(*!
<summary>
Beckhoff EL1008_EX: Extended 8-channel digital input terminal with diagnostics.
</summary>
<description>
Extends EL1008 with EtherCAT Working Counter and slave state diagnostics. Note: Simple digital terminals do
not feature CoE mailbox, hence ADS address is not present.
When used for I/O, link located fields or their containing buffers to the matching selected PDOs.
The record is not a packed wire buffer; compiler padding is not part of the device specification.
Unlinked/default values do not prove valid I/O. The caller evaluates bus/channel validity before use.
Use one owner task per instance and externally synchronize other access; multi-field snapshots are not atomic.
Copies store data without creating hardware links. Keep borrowed field references valid while consumers are bound.
This passive record performs no validation, synchronization, configuration or protocol advancement.
WcState=TRUE means process-data exchange is invalid. State is acyclic EtherCAT/link information,
not proof of current measurement validity. Link diagnostics to the matching slave InfoData entries.
The selected PDO representation is documented by the base terminal model.
InputToggle signals an input update by changing state; TRUE alone does not mean fresh data.
</description>
*)
TYPE EL1008_EX EXTENDS EL1008 :
STRUCT
	WcState AT %I* : BOOL;
	InputToggle AT %I* : BOOL;
	State AT %I* : UINT;
END_STRUCT
END_TYPE

// ---- DigitalIO/Outputs/EL2809/EL2809.TcDUT
(*
SPDX-FileCopyrightText: © 2026 Oleksandr Tiutyk <trofimich@gmail.com>
SPDX-License-Identifier: MIT
License: https://opensource.org/license/mit
*)

(*!
<summary>
Beckhoff EL2809: 16-channel HD digital output terminal (24 V DC, 0.5 A).
</summary>
<description>
Process image mapping structure for the high-density EL2809 16-channel discrete 24 V DC 0.5 A output terminal.
When used for I/O, link located fields or their containing buffers to the matching selected PDOs.
The record is not a packed wire buffer; compiler padding is not part of the device specification.
Unlinked/default values do not prove valid I/O. The caller evaluates bus/channel validity before use.
Use one owner task per instance and externally synchronize other access; multi-field snapshots are not atomic.
Copies store data without creating hardware links. Keep borrowed field references valid while consumers are bound.
This passive record performs no validation, synchronization, configuration or protocol advancement.
</description>
*)
TYPE EL2809 :
STRUCT
	Ch01 AT %Q* : BOOL;
	Ch02 AT %Q* : BOOL;
	Ch03 AT %Q* : BOOL;
	Ch04 AT %Q* : BOOL;
	Ch05 AT %Q* : BOOL;
	Ch06 AT %Q* : BOOL;
	Ch07 AT %Q* : BOOL;
	Ch08 AT %Q* : BOOL;
	Ch09 AT %Q* : BOOL;
	Ch10 AT %Q* : BOOL;
	Ch11 AT %Q* : BOOL;
	Ch12 AT %Q* : BOOL;
	Ch13 AT %Q* : BOOL;
	Ch14 AT %Q* : BOOL;
	Ch15 AT %Q* : BOOL;
	Ch16 AT %Q* : BOOL;
END_STRUCT
END_TYPE

// ---- DigitalIO/Outputs/EL2809/EL2809_EX.TcDUT
(*
SPDX-FileCopyrightText: © 2026 Oleksandr Tiutyk <trofimich@gmail.com>
SPDX-License-Identifier: MIT
License: https://opensource.org/license/mit
*)

(*!
<summary>
Beckhoff EL2809_EX: Extended 16-channel HD digital output terminal with diagnostics.
</summary>
<description>
Extends EL2809 with EtherCAT Working Counter and slave state diagnostics.
When used for I/O, link located fields or their containing buffers to the matching selected PDOs.
The record is not a packed wire buffer; compiler padding is not part of the device specification.
Unlinked/default values do not prove valid I/O. The caller evaluates bus/channel validity before use.
Use one owner task per instance and externally synchronize other access; multi-field snapshots are not atomic.
Copies store data without creating hardware links. Keep borrowed field references valid while consumers are bound.
This passive record performs no validation, synchronization, configuration or protocol advancement.
WcState=TRUE means process-data exchange is invalid. State is acyclic EtherCAT/link information,
not proof of current measurement validity. Link diagnostics to the matching slave InfoData entries.
The selected PDO representation is documented by the base terminal model.
</description>
*)
TYPE EL2809_EX EXTENDS EL2809 :
STRUCT
	WcState AT %I* : BOOL;
	State AT %I* : UINT;
END_STRUCT
END_TYPE

// ---- DigitalIO/Outputs/EL2622/EL2622.TcDUT
(*
SPDX-FileCopyrightText: © 2026 Oleksandr Tiutyk <trofimich@gmail.com>
SPDX-License-Identifier: MIT
License: https://opensource.org/license/mit
*)

(*!
<summary>
Beckhoff EL2622: 2-channel relay output terminal (230 V AC / 30 V DC, normally open make contacts).
</summary>
<description>
Process image mapping structure for the EL2622 potential-free relay output terminal.
Each channel switches up to 5 A AC/DC for resistive loads or 2 A AC/DC for inductive loads.
The terminal has two make contacts, not changeover contacts, and does not pass through power contacts.
When used for I/O, link located fields or their containing buffers to the matching selected PDOs.
The record is not a packed wire buffer; compiler padding is not part of the device specification.
Unlinked/default values do not prove valid I/O. The caller evaluates bus/channel validity before use.
Use one owner task per instance and externally synchronize other access; multi-field snapshots are not atomic.
Copies store data without creating hardware links. Keep borrowed field references valid while consumers are bound.
This passive record performs no validation, synchronization, configuration or protocol advancement.
</description>
*)
TYPE EL2622 :
STRUCT
	Ch1 AT %Q* : BOOL;
	Ch2 AT %Q* : BOOL;
END_STRUCT
END_TYPE

// ---- DigitalIO/Outputs/EL2622/EL2622_EX.TcDUT
(*
SPDX-FileCopyrightText: © 2026 Oleksandr Tiutyk <trofimich@gmail.com>
SPDX-License-Identifier: MIT
License: https://opensource.org/license/mit
*)

(*!
<summary>
Beckhoff EL2622_EX: Extended 2-channel relay output terminal with diagnostics.
</summary>
<description>
Extends EL2622 with EtherCAT Working Counter and slave state diagnostics.
Two make contacts are rated 230 V AC / 30 V DC, with 5 A resistive or 2 A inductive current per channel.
When used for I/O, link located fields or their containing buffers to the matching selected PDOs.
The record is not a packed wire buffer; compiler padding is not part of the device specification.
Unlinked/default values do not prove valid I/O. The caller evaluates bus/channel validity before use.
Use one owner task per instance and externally synchronize other access; multi-field snapshots are not atomic.
Copies store data without creating hardware links. Keep borrowed field references valid while consumers are bound.
This passive record performs no validation, synchronization, configuration or protocol advancement.
WcState=TRUE means process-data exchange is invalid. State is acyclic EtherCAT/link information,
not proof of current measurement validity. Link diagnostics to the matching slave InfoData entries.
The selected PDO representation is documented by the base terminal model.
</description>
*)
TYPE EL2622_EX EXTENDS EL2622 :
STRUCT
	WcState AT %I* : BOOL;
	State AT %I* : UINT;
END_STRUCT
END_TYPE

// ---- DigitalIO/Outputs/EL2624/EL2624.TcDUT
(*
SPDX-FileCopyrightText: © 2026 Oleksandr Tiutyk <trofimich@gmail.com>
SPDX-License-Identifier: MIT
License: https://opensource.org/license/mit
*)

(*!
<summary>
Beckhoff EL2624: 4-channel relay output terminal (125 V AC / 30 V DC, normally open make contacts).
</summary>
<description>
Process image mapping structure for the EL2624 potential-free relay output terminal.
Resistive switching ratings are 0.5 A AC at 125 V AC and 2 A DC at 30 V DC per channel.
When used for I/O, link located fields or their containing buffers to the matching selected PDOs.
The record is not a packed wire buffer; compiler padding is not part of the device specification.
Unlinked/default values do not prove valid I/O. The caller evaluates bus/channel validity before use.
Use one owner task per instance and externally synchronize other access; multi-field snapshots are not atomic.
Copies store data without creating hardware links. Keep borrowed field references valid while consumers are bound.
This passive record performs no validation, synchronization, configuration or protocol advancement.
</description>
*)
TYPE EL2624 :
STRUCT
	Ch1 AT %Q* : BOOL;
	Ch2 AT %Q* : BOOL;
	Ch3 AT %Q* : BOOL;
	Ch4 AT %Q* : BOOL;
END_STRUCT
END_TYPE

// ---- DigitalIO/Outputs/EL2624/EL2624_EX.TcDUT
(*
SPDX-FileCopyrightText: © 2026 Oleksandr Tiutyk <trofimich@gmail.com>
SPDX-License-Identifier: MIT
License: https://opensource.org/license/mit
*)

(*!
<summary>
Beckhoff EL2624_EX: Extended 4-channel relay output terminal with diagnostics.
</summary>
<description>
Extends EL2624 with EtherCAT Working Counter and slave state diagnostics.
Four make contacts are rated 125 V AC / 30 V DC, with 0.5 A AC / 2 A DC resistive current per channel.
When used for I/O, link located fields or their containing buffers to the matching selected PDOs.
The record is not a packed wire buffer; compiler padding is not part of the device specification.
Unlinked/default values do not prove valid I/O. The caller evaluates bus/channel validity before use.
Use one owner task per instance and externally synchronize other access; multi-field snapshots are not atomic.
Copies store data without creating hardware links. Keep borrowed field references valid while consumers are bound.
This passive record performs no validation, synchronization, configuration or protocol advancement.
WcState=TRUE means process-data exchange is invalid. State is acyclic EtherCAT/link information,
not proof of current measurement validity. Link diagnostics to the matching slave InfoData entries.
The selected PDO representation is documented by the base terminal model.
</description>
*)
TYPE EL2624_EX EXTENDS EL2624 :
STRUCT
	WcState AT %I* : BOOL;
	State AT %I* : UINT;
END_STRUCT
END_TYPE

// ---- Serial/EL6001/EL6001.TcDUT
(*
SPDX-FileCopyrightText: © 2026 Oleksandr Tiutyk <trofimich@gmail.com>
SPDX-License-Identifier: MIT
License: https://opensource.org/license/mit
*)

(*!
<summary>
Beckhoff EL6001: 1-channel serial interface terminal (RS232).
</summary>
<description>
Process image mapping structure for the EL6001 1-channel RS232 communication terminal.
When used for I/O, link located fields or their containing buffers to the matching selected PDOs.
The record is not a packed wire buffer; compiler padding is not part of the device specification.
Unlinked/default values do not prove valid I/O. The caller evaluates bus/channel validity before use.
Use one owner task per instance and externally synchronize other access; multi-field snapshots are not atomic.
Copies store data without creating hardware links. Keep borrowed field references valid while consumers are bound.
This passive record performs no validation, synchronization, configuration or protocol advancement.
Select the 22-byte serial payload with 16-bit status/control words; larger buffers and 9-bit modes
are outside this model. The owning service implements the transmit/receive toggle handshake.
</description>
*)
TYPE EL6001 :
STRUCT
	Ch1 : EL6001_CHANNEL;
END_STRUCT
END_TYPE

// ---- Serial/EL6001/EL6001_CHANNEL.TcDUT
(*
SPDX-FileCopyrightText: © 2026 Oleksandr Tiutyk <trofimich@gmail.com>
SPDX-License-Identifier: MIT
License: https://opensource.org/license/mit
*)

(*!
<summary>
Beckhoff EL6001: Serial RS232 communication channel process image.
</summary>
<description>
Encapsulates 22-byte input (InData) and output (OutData) process data for the EL6001 RS232 interface.
When used for I/O, link located fields or their containing buffers to the matching selected PDOs.
The record is not a packed wire buffer; compiler padding is not part of the device specification.
Unlinked/default values do not prove valid I/O. The caller evaluates bus/channel validity before use.
Use one owner task per instance and externally synchronize other access; multi-field snapshots are not atomic.
Copies store data without creating hardware links. Keep borrowed field references valid while consumers are bound.
This passive record performs no validation, synchronization, configuration or protocol advancement.
Select the 22-byte serial payload with 16-bit status/control words; larger buffers and 9-bit modes
are outside this model. The owning service implements the transmit/receive toggle handshake.
</description>
*)
TYPE EL6001_CHANNEL :
STRUCT
	InData AT %I* : EL6xxx22ByteInData;
	OutData AT %Q* : EL6xxx22ByteOutData;
END_STRUCT
END_TYPE

// ---- Serial/EL6001/EL6001_EX.TcDUT
(*
SPDX-FileCopyrightText: © 2026 Oleksandr Tiutyk <trofimich@gmail.com>
SPDX-License-Identifier: MIT
License: https://opensource.org/license/mit
*)

(*!
<summary>
Beckhoff EL6001_EX: Extended 1-channel serial interface terminal with diagnostics.
</summary>
<description>
Extends EL6001 with EtherCAT Working Counter, slave state, and CoE mailbox ADS address diagnostics.
When used for I/O, link located fields or their containing buffers to the matching selected PDOs.
The record is not a packed wire buffer; compiler padding is not part of the device specification.
Unlinked/default values do not prove valid I/O. The caller evaluates bus/channel validity before use.
Use one owner task per instance and externally synchronize other access; multi-field snapshots are not atomic.
Copies store data without creating hardware links. Keep borrowed field references valid while consumers are bound.
This passive record performs no validation, synchronization, configuration or protocol advancement.
WcState=TRUE means process-data exchange is invalid. State is acyclic EtherCAT/link information,
not proof of current measurement validity. Link diagnostics to the matching slave InfoData entries.
The selected PDO representation is documented by the base terminal model.
InputToggle signals an input update by changing state; TRUE alone does not mean fresh data.
AdsAddr is acyclic mailbox addressing information, not a measurement-validity indicator.
Select the 22-byte serial payload with 16-bit status/control words; larger buffers and 9-bit modes
are outside this model. The owning service implements the transmit/receive toggle handshake.
</description>
*)
TYPE EL6001_EX EXTENDS EL6001 :
STRUCT
	WcState AT %I* : BOOL;
	InputToggle AT %I* : BOOL;
	State AT %I* : UINT;
	AdsAddr AT %I* : Global.AMSADDR;
END_STRUCT
END_TYPE

// ---- Serial/EL6002/EL6002.TcDUT
(*
SPDX-FileCopyrightText: © 2026 Oleksandr Tiutyk <trofimich@gmail.com>
SPDX-License-Identifier: MIT
License: https://opensource.org/license/mit
*)

(*!
<summary>
Beckhoff EL6002: 2-channel serial interface terminal (RS232).
</summary>
<description>
Process image mapping structure for the EL6002 2-channel RS232 communication terminal.
When used for I/O, link located fields or their containing buffers to the matching selected PDOs.
The record is not a packed wire buffer; compiler padding is not part of the device specification.
Unlinked/default values do not prove valid I/O. The caller evaluates bus/channel validity before use.
Use one owner task per instance and externally synchronize other access; multi-field snapshots are not atomic.
Copies store data without creating hardware links. Keep borrowed field references valid while consumers are bound.
This passive record performs no validation, synchronization, configuration or protocol advancement.
Select the 22-byte serial payload with 16-bit status/control words; larger buffers and 9-bit modes
are outside this model. The owning service implements the transmit/receive toggle handshake.
</description>
*)
TYPE EL6002 :
STRUCT
	Ch1 : EL6002_CHANNEL;
	Ch2 : EL6002_CHANNEL;
END_STRUCT
END_TYPE

// ---- Serial/EL6002/EL6002_CHANNEL.TcDUT
(*
SPDX-FileCopyrightText: © 2026 Oleksandr Tiutyk <trofimich@gmail.com>
SPDX-License-Identifier: MIT
License: https://opensource.org/license/mit
*)

(*!
<summary>
Beckhoff EL6002: Serial RS232 communication channel process image.
</summary>
<description>
Encapsulates 22-byte input (InData) and output (OutData) process data for the EL6002 RS232 interface.
When used for I/O, link located fields or their containing buffers to the matching selected PDOs.
The record is not a packed wire buffer; compiler padding is not part of the device specification.
Unlinked/default values do not prove valid I/O. The caller evaluates bus/channel validity before use.
Use one owner task per instance and externally synchronize other access; multi-field snapshots are not atomic.
Copies store data without creating hardware links. Keep borrowed field references valid while consumers are bound.
This passive record performs no validation, synchronization, configuration or protocol advancement.
Select the 22-byte serial payload with 16-bit status/control words; larger buffers and 9-bit modes
are outside this model. The owning service implements the transmit/receive toggle handshake.
</description>
*)
TYPE EL6002_CHANNEL :
STRUCT
	InData AT %I* : EL6xxx22ByteInData;
	OutData AT %Q* : EL6xxx22ByteOutData;
END_STRUCT
END_TYPE

// ---- Serial/EL6002/EL6002_EX.TcDUT
(*
SPDX-FileCopyrightText: © 2026 Oleksandr Tiutyk <trofimich@gmail.com>
SPDX-License-Identifier: MIT
License: https://opensource.org/license/mit
*)

(*!
<summary>
Beckhoff EL6002_EX: Extended 2-channel serial interface terminal with diagnostics.
</summary>
<description>
Extends EL6002 with EtherCAT Working Counter, slave state, and CoE mailbox ADS address diagnostics.
When used for I/O, link located fields or their containing buffers to the matching selected PDOs.
The record is not a packed wire buffer; compiler padding is not part of the device specification.
Unlinked/default values do not prove valid I/O. The caller evaluates bus/channel validity before use.
Use one owner task per instance and externally synchronize other access; multi-field snapshots are not atomic.
Copies store data without creating hardware links. Keep borrowed field references valid while consumers are bound.
This passive record performs no validation, synchronization, configuration or protocol advancement.
WcState=TRUE means process-data exchange is invalid. State is acyclic EtherCAT/link information,
not proof of current measurement validity. Link diagnostics to the matching slave InfoData entries.
The selected PDO representation is documented by the base terminal model.
InputToggle signals an input update by changing state; TRUE alone does not mean fresh data.
AdsAddr is acyclic mailbox addressing information, not a measurement-validity indicator.
Select the 22-byte serial payload with 16-bit status/control words; larger buffers and 9-bit modes
are outside this model. The owning service implements the transmit/receive toggle handshake.
</description>
*)
TYPE EL6002_EX EXTENDS EL6002 :
STRUCT
	WcState AT %I* : BOOL;
	InputToggle AT %I* : BOOL;
	State AT %I* : UINT;
	AdsAddr AT %I* : Global.AMSADDR;
END_STRUCT
END_TYPE

// ---- Serial/EL6021/EL6021.TcDUT
(*
SPDX-FileCopyrightText: © 2026 Oleksandr Tiutyk <trofimich@gmail.com>
SPDX-License-Identifier: MIT
License: https://opensource.org/license/mit
*)

(*!
<summary>
Beckhoff EL6021: 1-channel serial interface terminal (RS422 / RS485).
</summary>
<description>
Process image mapping structure for the EL6021 1-channel RS422/RS485 communication terminal.
When used for I/O, link located fields or their containing buffers to the matching selected PDOs.
The record is not a packed wire buffer; compiler padding is not part of the device specification.
Unlinked/default values do not prove valid I/O. The caller evaluates bus/channel validity before use.
Use one owner task per instance and externally synchronize other access; multi-field snapshots are not atomic.
Copies store data without creating hardware links. Keep borrowed field references valid while consumers are bound.
This passive record performs no validation, synchronization, configuration or protocol advancement.
Select the 22-byte serial payload with 16-bit status/control words; larger buffers and 9-bit modes
are outside this model. The owning service implements the transmit/receive toggle handshake.
</description>
*)
TYPE EL6021 :
STRUCT
	Ch1 : EL6021_CHANNEL;
END_STRUCT
END_TYPE

// ---- Serial/EL6021/EL6021_CHANNEL.TcDUT
(*
SPDX-FileCopyrightText: © 2026 Oleksandr Tiutyk <trofimich@gmail.com>
SPDX-License-Identifier: MIT
License: https://opensource.org/license/mit
*)

(*!
<summary>
Beckhoff EL6021: Serial RS422/RS485 communication channel process image.
</summary>
<description>
Encapsulates 22-byte input (InData) and output (OutData) process data for the EL6021 RS422/RS485 interface.
When used for I/O, link located fields or their containing buffers to the matching selected PDOs.
The record is not a packed wire buffer; compiler padding is not part of the device specification.
Unlinked/default values do not prove valid I/O. The caller evaluates bus/channel validity before use.
Use one owner task per instance and externally synchronize other access; multi-field snapshots are not atomic.
Copies store data without creating hardware links. Keep borrowed field references valid while consumers are bound.
This passive record performs no validation, synchronization, configuration or protocol advancement.
Select the 22-byte serial payload with 16-bit status/control words; larger buffers and 9-bit modes
are outside this model. The owning service implements the transmit/receive toggle handshake.
</description>
*)
TYPE EL6021_CHANNEL :
STRUCT
	InData AT %I* : EL6xxx22ByteInData;
	OutData AT %Q* : EL6xxx22ByteOutData;
END_STRUCT
END_TYPE

// ---- Serial/EL6021/EL6021_EX.TcDUT
(*
SPDX-FileCopyrightText: © 2026 Oleksandr Tiutyk <trofimich@gmail.com>
SPDX-License-Identifier: MIT
License: https://opensource.org/license/mit
*)

(*!
<summary>
Beckhoff EL6021_EX: Extended 1-channel serial interface terminal with diagnostics.
</summary>
<description>
Extends EL6021 with EtherCAT Working Counter, slave state, and CoE mailbox ADS address diagnostics.
When used for I/O, link located fields or their containing buffers to the matching selected PDOs.
The record is not a packed wire buffer; compiler padding is not part of the device specification.
Unlinked/default values do not prove valid I/O. The caller evaluates bus/channel validity before use.
Use one owner task per instance and externally synchronize other access; multi-field snapshots are not atomic.
Copies store data without creating hardware links. Keep borrowed field references valid while consumers are bound.
This passive record performs no validation, synchronization, configuration or protocol advancement.
WcState=TRUE means process-data exchange is invalid. State is acyclic EtherCAT/link information,
not proof of current measurement validity. Link diagnostics to the matching slave InfoData entries.
The selected PDO representation is documented by the base terminal model.
InputToggle signals an input update by changing state; TRUE alone does not mean fresh data.
AdsAddr is acyclic mailbox addressing information, not a measurement-validity indicator.
Select the 22-byte serial payload with 16-bit status/control words; larger buffers and 9-bit modes
are outside this model. The owning service implements the transmit/receive toggle handshake.
</description>
*)
TYPE EL6021_EX EXTENDS EL6021 :
STRUCT
	WcState AT %I* : BOOL;
	InputToggle AT %I* : BOOL;
	State AT %I* : UINT;
	AdsAddr AT %I* : Global.AMSADDR;
END_STRUCT
END_TYPE

// ---- Counters/COUNTER_INPUT_CHANNEL.TcDUT
(*
SPDX-FileCopyrightText: © 2026 Oleksandr Tiutyk <trofimich@gmail.com>
SPDX-License-Identifier: MIT
License: https://opensource.org/license/mit
*)

(*!
<summary>
Beckhoff counter input channel process image.
</summary>
<description>
Encapsulates 16-bit status word and 32-bit unsigned counter value (CounterValue : UDINT) for fast counter
terminals.
When used for I/O, link located fields or their containing buffers to the matching selected PDOs.
The record is not a packed wire buffer; compiler padding is not part of the device specification.
Unlinked/default values do not prove valid I/O. The caller evaluates bus/channel validity before use.
Use one owner task per instance and externally synchronize other access; multi-field snapshots are not atomic.
Copies store data without creating hardware links. Keep borrowed field references valid while consumers are bound.
This passive record performs no validation, synchronization, configuration or protocol advancement.
</description>
*)
TYPE COUNTER_INPUT_CHANNEL :
STRUCT
	Status AT %I* : WORD;
	CounterValue AT %I* : UDINT;
END_STRUCT
END_TYPE

// ---- Counters/COUNTER_OUTPUT_CHANNEL.TcDUT
(*
SPDX-FileCopyrightText: © 2026 Oleksandr Tiutyk <trofimich@gmail.com>
SPDX-License-Identifier: MIT
License: https://opensource.org/license/mit
*)

(*!
<summary>
Beckhoff counter output control channel process image.
</summary>
<description>
Encapsulates 16-bit control word and 32-bit unsigned preset counter value (SetCounterValue : UDINT) for fast
counter terminals.
When used for I/O, link located fields or their containing buffers to the matching selected PDOs.
The record is not a packed wire buffer; compiler padding is not part of the device specification.
Unlinked/default values do not prove valid I/O. The caller evaluates bus/channel validity before use.
Use one owner task per instance and externally synchronize other access; multi-field snapshots are not atomic.
Copies store data without creating hardware links. Keep borrowed field references valid while consumers are bound.
This passive record performs no validation, synchronization, configuration or protocol advancement.
</description>
*)
TYPE COUNTER_OUTPUT_CHANNEL :
STRUCT
	Control AT %Q* : WORD;
	SetCounterValue AT %Q* : UDINT;
END_STRUCT
END_TYPE

// ---- Counters/COUNTER_CHANNEL.TcDUT
(*
SPDX-FileCopyrightText: © 2026 Oleksandr Tiutyk <trofimich@gmail.com>
SPDX-License-Identifier: MIT
License: https://opensource.org/license/mit
*)

(*!
<summary>
Beckhoff bidirectional counter channel process image.
</summary>
<description>
Aggregates input status/value (COUNTER_INPUT_CHANNEL) and output control/preset (COUNTER_OUTPUT_CHANNEL) for
one counter channel.
When used for I/O, link located fields or their containing buffers to the matching selected PDOs.
The record is not a packed wire buffer; compiler padding is not part of the device specification.
Unlinked/default values do not prove valid I/O. The caller evaluates bus/channel validity before use.
Use one owner task per instance and externally synchronize other access; multi-field snapshots are not atomic.
Copies store data without creating hardware links. Keep borrowed field references valid while consumers are bound.
This passive record performs no validation, synchronization, configuration or protocol advancement.
</description>
*)
TYPE COUNTER_CHANNEL :
STRUCT
	In : COUNTER_INPUT_CHANNEL;
	Out : COUNTER_OUTPUT_CHANNEL;
END_STRUCT
END_TYPE

// ---- Counters/EL1502/EL1502.TcDUT
(*
SPDX-FileCopyrightText: © 2026 Oleksandr Tiutyk <trofimich@gmail.com>
SPDX-License-Identifier: MIT
License: https://opensource.org/license/mit
*)

(*!
<summary>
Beckhoff EL1502: 2-channel up/down counter terminal (24 V DC, 100 kHz).
</summary>
<description>
Requires the 2Ch. Counter assignment: TxPDOs 0x1A00/0x1A01 and RxPDOs 0x1600/0x1601.
Each channel is a 32-bit counter with 16-bit status/control; direction is configured through CoE.
The factory 1Ch. +/- Counter assignment 0x1A02/0x1602 is not represented.
This model does not provide two independent hardware up/down input pairs.
When used for I/O, link located fields or their containing buffers to the matching selected PDOs.
The record is not a packed wire buffer; compiler padding is not part of the device specification.
Unlinked/default values do not prove valid I/O. The caller evaluates bus/channel validity before use.
Use one owner task per instance and externally synchronize other access; multi-field snapshots are not atomic.
Copies store data without creating hardware links. Keep borrowed field references valid while consumers are bound.
This passive record performs no validation, synchronization, configuration or protocol advancement.
</description>
*)
TYPE EL1502 :
STRUCT
	Ch1 : COUNTER_CHANNEL;
	Ch2 : COUNTER_CHANNEL;
END_STRUCT
END_TYPE

// ---- Counters/EL1502/EL1502_EX.TcDUT
(*
SPDX-FileCopyrightText: © 2026 Oleksandr Tiutyk <trofimich@gmail.com>
SPDX-License-Identifier: MIT
License: https://opensource.org/license/mit
*)

(*!
<summary>
Beckhoff EL1502_EX: Extended 2-channel counter terminal with diagnostics.
</summary>
<description>
Extends EL1502 with EtherCAT Working Counter, slave state, and CoE mailbox ADS address diagnostics.
When used for I/O, link located fields or their containing buffers to the matching selected PDOs.
The record is not a packed wire buffer; compiler padding is not part of the device specification.
Unlinked/default values do not prove valid I/O. The caller evaluates bus/channel validity before use.
Use one owner task per instance and externally synchronize other access; multi-field snapshots are not atomic.
Copies store data without creating hardware links. Keep borrowed field references valid while consumers are bound.
This passive record performs no validation, synchronization, configuration or protocol advancement.
WcState=TRUE means process-data exchange is invalid. State is acyclic EtherCAT/link information,
not proof of current measurement validity. Link diagnostics to the matching slave InfoData entries.
The selected PDO representation is documented by the base terminal model.
InputToggle signals an input update by changing state; TRUE alone does not mean fresh data.
AdsAddr is acyclic mailbox addressing information, not a measurement-validity indicator.
</description>
*)
TYPE EL1502_EX EXTENDS EL1502 :
STRUCT
	WcState AT %I* : BOOL;
	InputToggle AT %I* : BOOL;
	State AT %I* : UINT;
	AdsAddr AT %I* : Global.AMSADDR;
END_STRUCT
END_TYPE

// ---- Counters/EL1512/EL1512.TcDUT
(*
SPDX-FileCopyrightText: © 2026 Oleksandr Tiutyk <trofimich@gmail.com>
SPDX-License-Identifier: MIT
License: https://opensource.org/license/mit
*)

(*!
<summary>
Beckhoff EL1512: 2-channel up/down counter terminal (24 V DC).
</summary>
<description>
Represents the default 2Ch. Counter assignment: TxPDOs 0x1A00/0x1A01 and RxPDOs 0x1600/0x1601.
Each channel has 16-bit status/control and a 32-bit counter/preset. Direction is configured through CoE.
Single-channel up/down or gated-counter assignments are outside this model.
When used for I/O, link located fields or their containing buffers to the matching selected PDOs.
The record is not a packed wire buffer; compiler padding is not part of the device specification.
Unlinked/default values do not prove valid I/O. The caller evaluates bus/channel validity before use.
Use one owner task per instance and externally synchronize other access; multi-field snapshots are not atomic.
Copies store data without creating hardware links. Keep borrowed field references valid while consumers are bound.
This passive record performs no validation, synchronization, configuration or protocol advancement.
</description>
*)
TYPE EL1512 :
STRUCT
	Ch1 : COUNTER_CHANNEL;
	Ch2 : COUNTER_CHANNEL;
END_STRUCT
END_TYPE

// ---- Counters/EL1512/EL1512_EX.TcDUT
(*
SPDX-FileCopyrightText: © 2026 Oleksandr Tiutyk <trofimich@gmail.com>
SPDX-License-Identifier: MIT
License: https://opensource.org/license/mit
*)

(*!
<summary>
Beckhoff EL1512_EX: Extended 2-channel counter terminal with diagnostics.
</summary>
<description>
Extends EL1512 with EtherCAT Working Counter, slave state, and CoE mailbox ADS address diagnostics.
When used for I/O, link located fields or their containing buffers to the matching selected PDOs.
The record is not a packed wire buffer; compiler padding is not part of the device specification.
Unlinked/default values do not prove valid I/O. The caller evaluates bus/channel validity before use.
Use one owner task per instance and externally synchronize other access; multi-field snapshots are not atomic.
Copies store data without creating hardware links. Keep borrowed field references valid while consumers are bound.
This passive record performs no validation, synchronization, configuration or protocol advancement.
WcState=TRUE means process-data exchange is invalid. State is acyclic EtherCAT/link information,
not proof of current measurement validity. Link diagnostics to the matching slave InfoData entries.
The selected PDO representation is documented by the base terminal model.
InputToggle signals an input update by changing state; TRUE alone does not mean fresh data.
AdsAddr is acyclic mailbox addressing information, not a measurement-validity indicator.
</description>
*)
TYPE EL1512_EX EXTENDS EL1512 :
STRUCT
	WcState AT %I* : BOOL;
	InputToggle AT %I* : BOOL;
	State AT %I* : UINT;
	AdsAddr AT %I* : Global.AMSADDR;
END_STRUCT
END_TYPE

// ---- Encoders/INCREMENTAL_ENCODER_INPUT_CHANNEL.TcDUT
(*
SPDX-FileCopyrightText: © 2026 Oleksandr Tiutyk <trofimich@gmail.com>
SPDX-License-Identifier: MIT
License: https://opensource.org/license/mit
*)

(*!
<summary>
Beckhoff incremental encoder input channel process image.
</summary>
<description>
Encapsulates 16-bit status word, 32-bit position value, and 32-bit captured latch value.
Use the matching 32-bit main PDO of EL5101 enhanced mode or EL5151. EL5152 has no latch and uses
INCREMENTAL_ENCODER_COUNTER_INPUT_CHANNEL instead; 16-bit process images are unsupported.
When used for I/O, link located fields or their containing buffers to the matching selected PDOs.
The record is not a packed wire buffer; compiler padding is not part of the device specification.
Unlinked/default values do not prove valid I/O. The caller evaluates bus/channel validity before use.
Use one owner task per instance and externally synchronize other access; multi-field snapshots are not atomic.
Copies store data without creating hardware links. Keep borrowed field references valid while consumers are bound.
This passive record performs no validation, synchronization, configuration or protocol advancement.
</description>
*)
TYPE INCREMENTAL_ENCODER_INPUT_CHANNEL :
STRUCT
	Status AT %I* : WORD;
	Value AT %I* : UDINT;
	Latch AT %I* : UDINT;
END_STRUCT
END_TYPE

// ---- Encoders/INCREMENTAL_ENCODER_OUTPUT_CHANNEL.TcDUT
(*
SPDX-FileCopyrightText: © 2026 Oleksandr Tiutyk <trofimich@gmail.com>
SPDX-License-Identifier: MIT
License: https://opensource.org/license/mit
*)

(*!
<summary>
Beckhoff incremental encoder output channel process image.
</summary>
<description>
Encapsulates 16-bit control word and 32-bit preset position value.
When used for I/O, link located fields or their containing buffers to the matching selected PDOs.
The record is not a packed wire buffer; compiler padding is not part of the device specification.
Unlinked/default values do not prove valid I/O. The caller evaluates bus/channel validity before use.
Use one owner task per instance and externally synchronize other access; multi-field snapshots are not atomic.
Copies store data without creating hardware links. Keep borrowed field references valid while consumers are bound.
This passive record performs no validation, synchronization, configuration or protocol advancement.
</description>
*)
TYPE INCREMENTAL_ENCODER_OUTPUT_CHANNEL :
STRUCT
	Control AT %Q* : WORD;
	SetValue AT %Q* : UDINT;
END_STRUCT
END_TYPE

// ---- Encoders/INCREMENTAL_ENCODER_CHANNEL.TcDUT
(*
SPDX-FileCopyrightText: © 2026 Oleksandr Tiutyk <trofimich@gmail.com>
SPDX-License-Identifier: MIT
License: https://opensource.org/license/mit
*)

(*!
<summary>
Beckhoff bidirectional incremental encoder channel process image.
</summary>
<description>
Aggregates input position/status/latch and output control/preset for an incremental encoder interface.
Requires the matching 32-bit EL5101 enhanced or EL5151 main PDOs. EL5152 uses the latch-free
INCREMENTAL_ENCODER_COUNTER_CHANNEL; do not substitute these channel types for each other.
When used for I/O, link located fields or their containing buffers to the matching selected PDOs.
The record is not a packed wire buffer; compiler padding is not part of the device specification.
Unlinked/default values do not prove valid I/O. The caller evaluates bus/channel validity before use.
Use one owner task per instance and externally synchronize other access; multi-field snapshots are not atomic.
Copies store data without creating hardware links. Keep borrowed field references valid while consumers are bound.
This passive record performs no validation, synchronization, configuration or protocol advancement.
</description>
*)
TYPE INCREMENTAL_ENCODER_CHANNEL :
STRUCT
	In : INCREMENTAL_ENCODER_INPUT_CHANNEL;
	Out : INCREMENTAL_ENCODER_OUTPUT_CHANNEL;
END_STRUCT
END_TYPE

// ---- Encoders/INCREMENTAL_ENCODER_COUNTER_INPUT_CHANNEL.TcDUT
(*
SPDX-FileCopyrightText: © 2026 Oleksandr Tiutyk <trofimich@gmail.com>
SPDX-License-Identifier: MIT
License: https://opensource.org/license/mit
*)

(*!
<summary>Beckhoff EL5152 32-bit incremental encoder feedback without a latch.</summary>
<description>
Represents the 32-bit main input PDO for one EL5152 channel (0x1A00 or 0x1A04).
Status is 16-bit; Value is the 32-bit counter. This terminal has no latch value.
Optional period/frequency PDOs are outside this channel; disable them or link them separately.
Link fields individually and evaluate bus/channel validity before use; unlinked zeros are not valid data.
Use one owner task and externally synchronize other access. Copies are not atomic multi-field snapshots.
When used for I/O, link located fields or their containing buffers to the matching selected PDOs.
The record is not a packed wire buffer; compiler padding is not part of the device specification.
Unlinked/default values do not prove valid I/O. The caller evaluates bus/channel validity before use.
Use one owner task per instance and externally synchronize other access; multi-field snapshots are not atomic.
Copies store data without creating hardware links. Keep borrowed field references valid while consumers are bound.
This passive record performs no validation, synchronization, configuration or protocol advancement.
</description>
*)
TYPE INCREMENTAL_ENCODER_COUNTER_INPUT_CHANNEL :
STRUCT
	Status AT %I* : WORD;
	Value AT %I* : UDINT;
END_STRUCT
END_TYPE

// ---- Encoders/INCREMENTAL_ENCODER_COUNTER_CHANNEL.TcDUT
(*
SPDX-FileCopyrightText: © 2026 Oleksandr Tiutyk <trofimich@gmail.com>
SPDX-License-Identifier: MIT
License: https://opensource.org/license/mit
*)

(*!
<summary>Beckhoff EL5152 32-bit incremental encoder channel without a latch.</summary>
<description>
Combines a latch-free 32-bit counter input with the 16-bit control word and 32-bit counter preset.
Select the 32-bit main PDOs for the corresponding EL5152 channel; optional period/frequency PDOs are separate.
Link input and output fields individually; the aggregate is not a packed EtherCAT packet.
Use one owner task; externally synchronize other access. Copies store data without creating hardware links.
When used for I/O, link located fields or their containing buffers to the matching selected PDOs.
The record is not a packed wire buffer; compiler padding is not part of the device specification.
Unlinked/default values do not prove valid I/O. The caller evaluates bus/channel validity before use.
Use one owner task per instance and externally synchronize other access; multi-field snapshots are not atomic.
Copies store data without creating hardware links. Keep borrowed field references valid while consumers are bound.
This passive record performs no validation, synchronization, configuration or protocol advancement.
</description>
*)
TYPE INCREMENTAL_ENCODER_COUNTER_CHANNEL :
STRUCT
	In : INCREMENTAL_ENCODER_COUNTER_INPUT_CHANNEL;
	Out : INCREMENTAL_ENCODER_OUTPUT_CHANNEL;
END_STRUCT
END_TYPE

// ---- Encoders/SSI_ENCODER_CHANNEL.TcDUT
(*
SPDX-FileCopyrightText: © 2026 Oleksandr Tiutyk <trofimich@gmail.com>
SPDX-License-Identifier: MIT
License: https://opensource.org/license/mit
*)

(*!
<summary>
Beckhoff SSI absolute encoder channel process image.
</summary>
<description>
Represents the SSI 32-bit position and two-byte status variant.
EL5001 requires firmware 11 or later and selection of the two-byte status PDO (0x1A01).
Earlier EL5001 firmware supports only one status byte and is incompatible with this channel.
For EL5002 select the corresponding two-byte status PDO for each channel. No byte-status conversion occurs.
When used for I/O, link located fields or their containing buffers to the matching selected PDOs.
The record is not a packed wire buffer; compiler padding is not part of the device specification.
Unlinked/default values do not prove valid I/O. The caller evaluates bus/channel validity before use.
Use one owner task per instance and externally synchronize other access; multi-field snapshots are not atomic.
Copies store data without creating hardware links. Keep borrowed field references valid while consumers are bound.
This passive record performs no validation, synchronization, configuration or protocol advancement.
</description>
*)
TYPE SSI_ENCODER_CHANNEL :
STRUCT
	Status AT %I* : WORD;
	Value AT %I* : UDINT;
END_STRUCT
END_TYPE

// ---- Encoders/EL5101/EL5101.TcDUT
(*
SPDX-FileCopyrightText: © 2026 Oleksandr Tiutyk <trofimich@gmail.com>
SPDX-License-Identifier: MIT
License: https://opensource.org/license/mit
*)

(*!
<summary>
Beckhoff EL5101: 1-channel incremental encoder interface terminal (RS422 / TTL, 5 V / 24 V).
</summary>
<description>
Requires enhanced operating mode, available on EL5101 from firmware 14 / hardware 09,
and Standard 32-bit (MDP 511): TxPDO 0x1A04 and RxPDO 0x1603.
Ch1 contains 16-bit status/control and 32-bit counter, latch and preset values.
The normal 16-bit mode and optional frequency/period/timestamp PDOs are outside this model.
When used for I/O, link located fields or their containing buffers to the matching selected PDOs.
The record is not a packed wire buffer; compiler padding is not part of the device specification.
Unlinked/default values do not prove valid I/O. The caller evaluates bus/channel validity before use.
Use one owner task per instance and externally synchronize other access; multi-field snapshots are not atomic.
Copies store data without creating hardware links. Keep borrowed field references valid while consumers are bound.
This passive record performs no validation, synchronization, configuration or protocol advancement.
</description>
*)
TYPE EL5101 :
STRUCT
	Ch1 : INCREMENTAL_ENCODER_CHANNEL;
END_STRUCT
END_TYPE

// ---- Encoders/EL5101/EL5101_EX.TcDUT
(*
SPDX-FileCopyrightText: © 2026 Oleksandr Tiutyk <trofimich@gmail.com>
SPDX-License-Identifier: MIT
License: https://opensource.org/license/mit
*)

(*!
<summary>
Beckhoff EL5101_EX: Extended 1-channel incremental encoder terminal with diagnostics.
</summary>
<description>
Extends EL5101 with EtherCAT Working Counter, slave state, and CoE mailbox ADS address diagnostics.
When used for I/O, link located fields or their containing buffers to the matching selected PDOs.
The record is not a packed wire buffer; compiler padding is not part of the device specification.
Unlinked/default values do not prove valid I/O. The caller evaluates bus/channel validity before use.
Use one owner task per instance and externally synchronize other access; multi-field snapshots are not atomic.
Copies store data without creating hardware links. Keep borrowed field references valid while consumers are bound.
This passive record performs no validation, synchronization, configuration or protocol advancement.
WcState=TRUE means process-data exchange is invalid. State is acyclic EtherCAT/link information,
not proof of current measurement validity. Link diagnostics to the matching slave InfoData entries.
The selected PDO representation is documented by the base terminal model.
InputToggle signals an input update by changing state; TRUE alone does not mean fresh data.
AdsAddr is acyclic mailbox addressing information, not a measurement-validity indicator.
</description>
*)
TYPE EL5101_EX EXTENDS EL5101 :
STRUCT
	WcState AT %I* : BOOL;
	InputToggle AT %I* : BOOL;
	State AT %I* : UINT;
	AdsAddr AT %I* : Global.AMSADDR;
END_STRUCT
END_TYPE

// ---- Encoders/EL5151/EL5151.TcDUT
(*
SPDX-FileCopyrightText: © 2026 Oleksandr Tiutyk <trofimich@gmail.com>
SPDX-License-Identifier: MIT
License: https://opensource.org/license/mit
*)

(*!
<summary>
Beckhoff EL5151: 1-channel incremental encoder interface terminal (24 V HTL, single-ended).
</summary>
<description>
Represents Standard 32-bit (MDP 511) main PDOs: TxPDO 0x1A00 and RxPDO 0x1600.
Ch1 contains 16-bit status/control and 32-bit counter, latch and preset values.
Optional period/frequency/timestamp PDOs are outside this model; disable or link them separately.
The Standard 16-bit process image is unsupported.
When used for I/O, link located fields or their containing buffers to the matching selected PDOs.
The record is not a packed wire buffer; compiler padding is not part of the device specification.
Unlinked/default values do not prove valid I/O. The caller evaluates bus/channel validity before use.
Use one owner task per instance and externally synchronize other access; multi-field snapshots are not atomic.
Copies store data without creating hardware links. Keep borrowed field references valid while consumers are bound.
This passive record performs no validation, synchronization, configuration or protocol advancement.
</description>
*)
TYPE EL5151 :
STRUCT
	Ch1 : INCREMENTAL_ENCODER_CHANNEL;
END_STRUCT
END_TYPE

// ---- Encoders/EL5151/EL5151_EX.TcDUT
(*
SPDX-FileCopyrightText: © 2026 Oleksandr Tiutyk <trofimich@gmail.com>
SPDX-License-Identifier: MIT
License: https://opensource.org/license/mit
*)

(*!
<summary>
Beckhoff EL5151_EX: Extended 1-channel 24 V incremental encoder terminal with diagnostics.
</summary>
<description>
Extends EL5151 with EtherCAT Working Counter, slave state, and CoE mailbox ADS address diagnostics.
When used for I/O, link located fields or their containing buffers to the matching selected PDOs.
The record is not a packed wire buffer; compiler padding is not part of the device specification.
Unlinked/default values do not prove valid I/O. The caller evaluates bus/channel validity before use.
Use one owner task per instance and externally synchronize other access; multi-field snapshots are not atomic.
Copies store data without creating hardware links. Keep borrowed field references valid while consumers are bound.
This passive record performs no validation, synchronization, configuration or protocol advancement.
WcState=TRUE means process-data exchange is invalid. State is acyclic EtherCAT/link information,
not proof of current measurement validity. Link diagnostics to the matching slave InfoData entries.
The selected PDO representation is documented by the base terminal model.
InputToggle signals an input update by changing state; TRUE alone does not mean fresh data.
AdsAddr is acyclic mailbox addressing information, not a measurement-validity indicator.
</description>
*)
TYPE EL5151_EX EXTENDS EL5151 :
STRUCT
	WcState AT %I* : BOOL;
	InputToggle AT %I* : BOOL;
	State AT %I* : UINT;
	AdsAddr AT %I* : Global.AMSADDR;
END_STRUCT
END_TYPE

// ---- Encoders/EL5152/EL5152.TcDUT
(*
SPDX-FileCopyrightText: © 2026 Oleksandr Tiutyk <trofimich@gmail.com>
SPDX-License-Identifier: MIT
License: https://opensource.org/license/mit
*)

(*!
<summary>
Beckhoff EL5152: 2-channel incremental encoder interface terminal (24 V HTL, single-ended).
</summary>
<description>
Represents the 32-bit main PDOs: channel 1 uses 0x1A00/0x1600; channel 2 uses 0x1A04/0x1602.
Both channels expose counter feedback and preset without a latch. Select Standard 32-bit (MDP 511);
optional period/frequency PDOs included by the ESI preset are outside this model and must be linked
separately if retained. The Standard 16-bit image is unsupported. Link each field individually.
Evaluate bus/channel validity before use. Use one owner task and synchronize other access.
When used for I/O, link located fields or their containing buffers to the matching selected PDOs.
The record is not a packed wire buffer; compiler padding is not part of the device specification.
Unlinked/default values do not prove valid I/O. The caller evaluates bus/channel validity before use.
Use one owner task per instance and externally synchronize other access; multi-field snapshots are not atomic.
Copies store data without creating hardware links. Keep borrowed field references valid while consumers are bound.
This passive record performs no validation, synchronization, configuration or protocol advancement.
</description>
*)
TYPE EL5152 :
STRUCT
	Ch1 : INCREMENTAL_ENCODER_COUNTER_CHANNEL;
	Ch2 : INCREMENTAL_ENCODER_COUNTER_CHANNEL;
END_STRUCT
END_TYPE

// ---- Encoders/EL5152/EL5152_EX.TcDUT
(*
SPDX-FileCopyrightText: © 2026 Oleksandr Tiutyk <trofimich@gmail.com>
SPDX-License-Identifier: MIT
License: https://opensource.org/license/mit
*)

(*!
<summary>
Beckhoff EL5152_EX: Extended 2-channel 24 V incremental encoder terminal with diagnostics.
</summary>
<description>
Extends EL5152 with EtherCAT Working Counter, slave state, and CoE mailbox ADS address diagnostics.
When used for I/O, link located fields or their containing buffers to the matching selected PDOs.
The record is not a packed wire buffer; compiler padding is not part of the device specification.
Unlinked/default values do not prove valid I/O. The caller evaluates bus/channel validity before use.
Use one owner task per instance and externally synchronize other access; multi-field snapshots are not atomic.
Copies store data without creating hardware links. Keep borrowed field references valid while consumers are bound.
This passive record performs no validation, synchronization, configuration or protocol advancement.
WcState=TRUE means process-data exchange is invalid. State is acyclic EtherCAT/link information,
not proof of current measurement validity. Link diagnostics to the matching slave InfoData entries.
The selected PDO representation is documented by the base terminal model.
InputToggle signals an input update by changing state; TRUE alone does not mean fresh data.
AdsAddr is acyclic mailbox addressing information, not a measurement-validity indicator.
</description>
*)
TYPE EL5152_EX EXTENDS EL5152 :
STRUCT
	WcState AT %I* : BOOL;
	InputToggle AT %I* : BOOL;
	State AT %I* : UINT;
	AdsAddr AT %I* : Global.AMSADDR;
END_STRUCT
END_TYPE

// ---- Encoders/EL5001/EL5001.TcDUT
(*
SPDX-FileCopyrightText: © 2026 Oleksandr Tiutyk <trofimich@gmail.com>
SPDX-License-Identifier: MIT
License: https://opensource.org/license/mit
*)

(*!
<summary>
Beckhoff EL5001: 1-channel SSI absolute encoder interface terminal.
</summary>
<description>
Process image mapping structure for the EL5001 synchronous serial interface (SSI) absolute encoder terminal.
Requires firmware 11 or later and the two-byte status PDO 0x1A01. The one-byte variant is unsupported.
When used for I/O, link located fields or their containing buffers to the matching selected PDOs.
The record is not a packed wire buffer; compiler padding is not part of the device specification.
Unlinked/default values do not prove valid I/O. The caller evaluates bus/channel validity before use.
Use one owner task per instance and externally synchronize other access; multi-field snapshots are not atomic.
Copies store data without creating hardware links. Keep borrowed field references valid while consumers are bound.
This passive record performs no validation, synchronization, configuration or protocol advancement.
</description>
*)
TYPE EL5001 :
STRUCT
	Ch1 : SSI_ENCODER_CHANNEL;
END_STRUCT
END_TYPE

// ---- Encoders/EL5001/EL5001_EX.TcDUT
(*
SPDX-FileCopyrightText: © 2026 Oleksandr Tiutyk <trofimich@gmail.com>
SPDX-License-Identifier: MIT
License: https://opensource.org/license/mit
*)

(*!
<summary>
Beckhoff EL5001_EX: Extended 1-channel SSI encoder terminal with diagnostics.
</summary>
<description>
Extends EL5001 with EtherCAT Working Counter, slave state, and CoE mailbox ADS address diagnostics.
When used for I/O, link located fields or their containing buffers to the matching selected PDOs.
The record is not a packed wire buffer; compiler padding is not part of the device specification.
Unlinked/default values do not prove valid I/O. The caller evaluates bus/channel validity before use.
Use one owner task per instance and externally synchronize other access; multi-field snapshots are not atomic.
Copies store data without creating hardware links. Keep borrowed field references valid while consumers are bound.
This passive record performs no validation, synchronization, configuration or protocol advancement.
WcState=TRUE means process-data exchange is invalid. State is acyclic EtherCAT/link information,
not proof of current measurement validity. Link diagnostics to the matching slave InfoData entries.
The selected PDO representation is documented by the base terminal model.
InputToggle signals an input update by changing state; TRUE alone does not mean fresh data.
AdsAddr is acyclic mailbox addressing information, not a measurement-validity indicator.
</description>
*)
TYPE EL5001_EX EXTENDS EL5001 :
STRUCT
	WcState AT %I* : BOOL;
	InputToggle AT %I* : BOOL;
	State AT %I* : UINT;
	AdsAddr AT %I* : Global.AMSADDR;
END_STRUCT
END_TYPE

// ---- Encoders/EL5002/EL5002.TcDUT
(*
SPDX-FileCopyrightText: © 2026 Oleksandr Tiutyk <trofimich@gmail.com>
SPDX-License-Identifier: MIT
License: https://opensource.org/license/mit
*)

(*!
<summary>
Beckhoff EL5002: 2-channel SSI absolute encoder interface terminal.
</summary>
<description>
Process image mapping structure for the EL5002 2-channel synchronous serial interface (SSI) absolute encoder
terminal.
Select the two-byte status PDO for each channel. The one-byte status variant is unsupported.
When used for I/O, link located fields or their containing buffers to the matching selected PDOs.
The record is not a packed wire buffer; compiler padding is not part of the device specification.
Unlinked/default values do not prove valid I/O. The caller evaluates bus/channel validity before use.
Use one owner task per instance and externally synchronize other access; multi-field snapshots are not atomic.
Copies store data without creating hardware links. Keep borrowed field references valid while consumers are bound.
This passive record performs no validation, synchronization, configuration or protocol advancement.
</description>
*)
TYPE EL5002 :
STRUCT
	Ch1 : SSI_ENCODER_CHANNEL;
	Ch2 : SSI_ENCODER_CHANNEL;
END_STRUCT
END_TYPE

// ---- Encoders/EL5002/EL5002_EX.TcDUT
(*
SPDX-FileCopyrightText: © 2026 Oleksandr Tiutyk <trofimich@gmail.com>
SPDX-License-Identifier: MIT
License: https://opensource.org/license/mit
*)

(*!
<summary>
Beckhoff EL5002_EX: Extended 2-channel SSI encoder terminal with diagnostics.
</summary>
<description>
Extends EL5002 with EtherCAT Working Counter, slave state, and CoE mailbox ADS address diagnostics.
When used for I/O, link located fields or their containing buffers to the matching selected PDOs.
The record is not a packed wire buffer; compiler padding is not part of the device specification.
Unlinked/default values do not prove valid I/O. The caller evaluates bus/channel validity before use.
Use one owner task per instance and externally synchronize other access; multi-field snapshots are not atomic.
Copies store data without creating hardware links. Keep borrowed field references valid while consumers are bound.
This passive record performs no validation, synchronization, configuration or protocol advancement.
WcState=TRUE means process-data exchange is invalid. State is acyclic EtherCAT/link information,
not proof of current measurement validity. Link diagnostics to the matching slave InfoData entries.
The selected PDO representation is documented by the base terminal model.
InputToggle signals an input update by changing state; TRUE alone does not mean fresh data.
AdsAddr is acyclic mailbox addressing information, not a measurement-validity indicator.
</description>
*)
TYPE EL5002_EX EXTENDS EL5002 :
STRUCT
	WcState AT %I* : BOOL;
	InputToggle AT %I* : BOOL;
	State AT %I* : UINT;
	AdsAddr AT %I* : Global.AMSADDR;
END_STRUCT
END_TYPE

// ---- PWM/PWM_OUTPUT_CHANNEL.TcDUT
(*
SPDX-FileCopyrightText: © 2026 Oleksandr Tiutyk <trofimich@gmail.com>
SPDX-License-Identifier: MIT
License: https://opensource.org/license/mit
*)

(*!
<summary>
Beckhoff PWM output channel process image.
</summary>
<description>
Represents the duty-only EL2502 standard PWM PDO with signed presentation selected through CoE.
DutyCycle 0..32767 represents 0..100 percent before user scaling; frequency is configured acyclically.
Cyclic-period and unsigned-presentation variants are outside this channel. No clamping or CoE configuration occurs.
When used for I/O, link located fields or their containing buffers to the matching selected PDOs.
The record is not a packed wire buffer; compiler padding is not part of the device specification.
Unlinked/default values do not prove valid I/O. The caller evaluates bus/channel validity before use.
Use one owner task per instance and externally synchronize other access; multi-field snapshots are not atomic.
Copies store data without creating hardware links. Keep borrowed field references valid while consumers are bound.
This passive record performs no validation, synchronization, configuration or protocol advancement.
</description>
*)
TYPE PWM_OUTPUT_CHANNEL :
STRUCT
	DutyCycle AT %Q* : INT;
END_STRUCT
END_TYPE

// ---- PWM/PULSE_TRAIN_INPUT_CHANNEL.TcDUT
(*
SPDX-FileCopyrightText: © 2026 Oleksandr Tiutyk <trofimich@gmail.com>
SPDX-License-Identifier: MIT
License: https://opensource.org/license/mit
*)

(*!
<summary>
Beckhoff pulse train output feedback status process image.
</summary>
<description>
Requires EL2521 Standard 32-bit (MDP 253/511), TxPDOs 0x1A01 and 0x1A05.
Status and CounterStatus belong to separate PDOs; both carry sync error at bit 13 and toggle at bit 15.
Status bit 6 reports a PTO error. Evaluate bus validity and both status words before using CounterValue.
Link each input field individually; zero values do not prove valid links. Legacy and 16-bit layouts are unsupported.
Use one owner task and externally synchronize other access; copies are not atomic multi-field snapshots.
When used for I/O, link located fields or their containing buffers to the matching selected PDOs.
The record is not a packed wire buffer; compiler padding is not part of the device specification.
Unlinked/default values do not prove valid I/O. The caller evaluates bus/channel validity before use.
Use one owner task per instance and externally synchronize other access; multi-field snapshots are not atomic.
Copies store data without creating hardware links. Keep borrowed field references valid while consumers are bound.
This passive record performs no validation, synchronization, configuration or protocol advancement.
</description>
*)
TYPE PULSE_TRAIN_INPUT_CHANNEL :
STRUCT
	Status AT %I* : WORD;
	//! <summary>ENC status from 0x1A05: counter-set acknowledgement bit 2, underflow 3 and overflow 4.</summary>
	CounterStatus AT %I* : WORD;
	//! <summary>32-bit feedback at 0x6020:11 from ENC Status PDO 0x1A05.</summary>
	CounterValue AT %I* : UDINT;
END_STRUCT
END_TYPE

// ---- PWM/PULSE_TRAIN_OUTPUT_CHANNEL.TcDUT
(*
SPDX-FileCopyrightText: © 2026 Oleksandr Tiutyk <trofimich@gmail.com>
SPDX-License-Identifier: MIT
License: https://opensource.org/license/mit
*)

(*!
<summary>
Beckhoff pulse train output command process image.
</summary>
<description>
Requires EL2521 enhanced mode, Standard 32-bit (MDP 253/511): RxPDOs 0x1601, 0x1607 and 0x1605.
Control bits 0, 1 and 2 select the base frequency, disable the ramp and start target travel.
Frequency preserves the UINT16 PDO bit pattern, including direction encoding selected through CoE.
In relative mode the interpreted command scales the selected base frequency by 1/32767; in direct mode
CoE 0x8010:16 multiplies the interpreted command in 0.01 Hz units. Frequency is not a 32-bit Hz value.
TargetCounterValue is a separate 32-bit target; SetCounterValue presets encoder feedback.
Link fields individually; this aggregate is not a packed wire buffer. Configure CoE before enabling outputs.
Use one owner task; externally synchronize other access. Copies do not create links or an atomic snapshot.
When used for I/O, link located fields or their containing buffers to the matching selected PDOs.
The record is not a packed wire buffer; compiler padding is not part of the device specification.
Unlinked/default values do not prove valid I/O. The caller evaluates bus/channel validity before use.
Use one owner task per instance and externally synchronize other access; multi-field snapshots are not atomic.
Copies store data without creating hardware links. Keep borrowed field references valid while consumers are bound.
This passive record performs no validation, synchronization, configuration or protocol advancement.
</description>
*)
TYPE PULSE_TRAIN_OUTPUT_CHANNEL :
STRUCT
	Control AT %Q* : WORD;
	//! <summary>Raw frequency command at 0x7010:11; interpretation follows CoE scaling and sign representation.</summary>
	Frequency AT %Q* : UINT;
	//! <summary>32-bit target at 0x7010:12, transmitted by PTO Target PDO 0x1607.</summary>
	TargetCounterValue AT %Q* : UDINT;
	//! <summary>ENC control from PDO 0x1605; bit 2 requests setting the feedback counter.</summary>
	CounterControl AT %Q* : WORD;
	//! <summary>Counter preset at 0x7020:11, accepted through CounterControl bit 2.</summary>
	SetCounterValue AT %Q* : UDINT;
END_STRUCT
END_TYPE

// ---- PWM/PULSE_TRAIN_CHANNEL.TcDUT
(*
SPDX-FileCopyrightText: © 2026 Oleksandr Tiutyk <trofimich@gmail.com>
SPDX-License-Identifier: MIT
License: https://opensource.org/license/mit
*)

(*!
<summary>
Beckhoff bidirectional pulse train channel process image.
</summary>
<description>
Combines EL2521 Standard 32-bit (MDP 253/511) input and output endpoints.
Select TxPDOs 0x1A01/0x1A05 and RxPDOs 0x1601/0x1607/0x1605 in enhanced operating mode.
Includes a 16-bit frequency command, 32-bit target, counter feedback and counter preset.
Link input and output fields individually; the aggregate is not one contiguous EtherCAT packet.
Use one owner task; synchronize external access. Copying stores data without creating new hardware links.
When used for I/O, link located fields or their containing buffers to the matching selected PDOs.
The record is not a packed wire buffer; compiler padding is not part of the device specification.
Unlinked/default values do not prove valid I/O. The caller evaluates bus/channel validity before use.
Use one owner task per instance and externally synchronize other access; multi-field snapshots are not atomic.
Copies store data without creating hardware links. Keep borrowed field references valid while consumers are bound.
This passive record performs no validation, synchronization, configuration or protocol advancement.
</description>
*)
TYPE PULSE_TRAIN_CHANNEL :
STRUCT
	In : PULSE_TRAIN_INPUT_CHANNEL;
	Out : PULSE_TRAIN_OUTPUT_CHANNEL;
END_STRUCT
END_TYPE

// ---- PWM/EL2502/EL2502.TcDUT
(*
SPDX-FileCopyrightText: © 2026 Oleksandr Tiutyk <trofimich@gmail.com>
SPDX-License-Identifier: MIT
License: https://opensource.org/license/mit
*)

(*!
<summary>
Beckhoff EL2502: 2-channel PWM output terminal (24 V DC, up to 20 kHz).
</summary>
<description>
Requires the duty-only Pulse width (standard) assignment, RxPDOs 0x1600 and 0x1601,
with signed presentation selected through CoE. Configure period/frequency before enabling outputs.
Cyclic-period and unsigned-presentation variants are outside this model.
When used for I/O, link located fields or their containing buffers to the matching selected PDOs.
The record is not a packed wire buffer; compiler padding is not part of the device specification.
Unlinked/default values do not prove valid I/O. The caller evaluates bus/channel validity before use.
Use one owner task per instance and externally synchronize other access; multi-field snapshots are not atomic.
Copies store data without creating hardware links. Keep borrowed field references valid while consumers are bound.
This passive record performs no validation, synchronization, configuration or protocol advancement.
</description>
*)
TYPE EL2502 :
STRUCT
	Ch1 : PWM_OUTPUT_CHANNEL;
	Ch2 : PWM_OUTPUT_CHANNEL;
END_STRUCT
END_TYPE

// ---- PWM/EL2502/EL2502_EX.TcDUT
(*
SPDX-FileCopyrightText: © 2026 Oleksandr Tiutyk <trofimich@gmail.com>
SPDX-License-Identifier: MIT
License: https://opensource.org/license/mit
*)

(*!
<summary>
Beckhoff EL2502_EX: Extended 2-channel PWM output terminal with diagnostics.
</summary>
<description>
Extends EL2502 with EtherCAT Working Counter, slave state, and CoE mailbox ADS address diagnostics. Note:
Output terminal does not feature InputToggle.
When used for I/O, link located fields or their containing buffers to the matching selected PDOs.
The record is not a packed wire buffer; compiler padding is not part of the device specification.
Unlinked/default values do not prove valid I/O. The caller evaluates bus/channel validity before use.
Use one owner task per instance and externally synchronize other access; multi-field snapshots are not atomic.
Copies store data without creating hardware links. Keep borrowed field references valid while consumers are bound.
This passive record performs no validation, synchronization, configuration or protocol advancement.
WcState=TRUE means process-data exchange is invalid. State is acyclic EtherCAT/link information,
not proof of current measurement validity. Link diagnostics to the matching slave InfoData entries.
The selected PDO representation is documented by the base terminal model.
AdsAddr is acyclic mailbox addressing information, not a measurement-validity indicator.
</description>
*)
TYPE EL2502_EX EXTENDS EL2502 :
STRUCT
	WcState AT %I* : BOOL;
	State AT %I* : UINT;
	AdsAddr AT %I* : Global.AMSADDR;
END_STRUCT
END_TYPE

// ---- PWM/EL2521/EL2521.TcDUT
(*
SPDX-FileCopyrightText: © 2026 Oleksandr Tiutyk <trofimich@gmail.com>
SPDX-License-Identifier: MIT
License: https://opensource.org/license/mit
*)

(*!
<summary>
Beckhoff EL2521: 1-channel pulse train output terminal (pulse/direction, up to 500 kHz).
</summary>
<description>
Requires enhanced operating mode (firmware 03 / hardware 02 or later supporting this preset)
and Predefined PDO Assignment Standard 32-bit (MDP 253/511).
Ch1 covers TxPDOs 0x1A01/0x1A05 and RxPDOs 0x1601/0x1607/0x1605.
Frequency remains a raw 16-bit command; target, counter feedback and counter preset are 32-bit.
Legacy and Standard 16-bit images are unsupported. Link each field separately and evaluate input validity.
Use one owner task; externally synchronize other access. Copies are data, not new links or atomic snapshots.
When used for I/O, link located fields or their containing buffers to the matching selected PDOs.
The record is not a packed wire buffer; compiler padding is not part of the device specification.
Unlinked/default values do not prove valid I/O. The caller evaluates bus/channel validity before use.
Use one owner task per instance and externally synchronize other access; multi-field snapshots are not atomic.
Copies store data without creating hardware links. Keep borrowed field references valid while consumers are bound.
This passive record performs no validation, synchronization, configuration or protocol advancement.
</description>
*)
TYPE EL2521 :
STRUCT
	Ch1 : PULSE_TRAIN_CHANNEL;
END_STRUCT
END_TYPE

// ---- PWM/EL2521/EL2521_EX.TcDUT
(*
SPDX-FileCopyrightText: © 2026 Oleksandr Tiutyk <trofimich@gmail.com>
SPDX-License-Identifier: MIT
License: https://opensource.org/license/mit
*)

(*!
<summary>
Beckhoff EL2521_EX: Extended 1-channel pulse train terminal with diagnostics.
</summary>
<description>
Extends EL2521 with EtherCAT Working Counter, slave state, and CoE mailbox ADS address diagnostics.
When used for I/O, link located fields or their containing buffers to the matching selected PDOs.
The record is not a packed wire buffer; compiler padding is not part of the device specification.
Unlinked/default values do not prove valid I/O. The caller evaluates bus/channel validity before use.
Use one owner task per instance and externally synchronize other access; multi-field snapshots are not atomic.
Copies store data without creating hardware links. Keep borrowed field references valid while consumers are bound.
This passive record performs no validation, synchronization, configuration or protocol advancement.
WcState=TRUE means process-data exchange is invalid. State is acyclic EtherCAT/link information,
not proof of current measurement validity. Link diagnostics to the matching slave InfoData entries.
The selected PDO representation is documented by the base terminal model.
InputToggle signals an input update by changing state; TRUE alone does not mean fresh data.
AdsAddr is acyclic mailbox addressing information, not a measurement-validity indicator.
</description>
*)
TYPE EL2521_EX EXTENDS EL2521 :
STRUCT
	WcState AT %I* : BOOL;
	InputToggle AT %I* : BOOL;
	State AT %I* : UINT;
	AdsAddr AT %I* : Global.AMSADDR;
END_STRUCT
END_TYPE

// ---- AnalogIO/Inputs/EL3051/EL3051.TcDUT
(*
SPDX-FileCopyrightText: © 2026 Oleksandr Tiutyk <trofimich@gmail.com>
SPDX-License-Identifier: MIT
License: https://opensource.org/license/mit
*)

(*!
<summary>
Beckhoff EL3051: 1-channel analog input terminal (4 .. 20 mA, 12-bit single-ended).
</summary>
<description>
Process image mapping structure for the EL3051 EtherCAT terminal with 1 analog input channel(s).
When used for I/O, link located fields or their containing buffers to the matching selected PDOs.
The record is not a packed wire buffer; compiler padding is not part of the device specification.
Unlinked/default values do not prove valid I/O. The caller evaluates bus/channel validity before use.
Use one owner task per instance and externally synchronize other access; multi-field snapshots are not atomic.
Copies store data without creating hardware links. Keep borrowed field references valid while consumers are bound.
This passive record performs no validation, synchronization, configuration or protocol advancement.
Select standard status-plus-value PDOs matching the declared Value type; compact value-only PDOs
are outside this model. Configure electrical range and scaling separately on the device.
</description>
*)
TYPE EL3051 :
STRUCT
	Ch1 : ANALOG_INPUT_INT_CHANNEL;
END_STRUCT
END_TYPE

// ---- AnalogIO/Inputs/EL3051/EL3051_EX.TcDUT
(*
SPDX-FileCopyrightText: © 2026 Oleksandr Tiutyk <trofimich@gmail.com>
SPDX-License-Identifier: MIT
License: https://opensource.org/license/mit
*)

(*!
<summary>
Beckhoff EL3051_EX: Extended 1-channel analog input terminal (4 .. 20 mA, 12-bit single-ended) with
diagnostics.
</summary>
<description>
Extends EL3051 with EtherCAT Working Counter, slave state, and CoE mailbox ADS address diagnostics.
When used for I/O, link located fields or their containing buffers to the matching selected PDOs.
The record is not a packed wire buffer; compiler padding is not part of the device specification.
Unlinked/default values do not prove valid I/O. The caller evaluates bus/channel validity before use.
Use one owner task per instance and externally synchronize other access; multi-field snapshots are not atomic.
Copies store data without creating hardware links. Keep borrowed field references valid while consumers are bound.
This passive record performs no validation, synchronization, configuration or protocol advancement.
WcState=TRUE means process-data exchange is invalid. State is acyclic EtherCAT/link information,
not proof of current measurement validity. Link diagnostics to the matching slave InfoData entries.
The selected PDO representation is documented by the base terminal model.
InputToggle signals an input update by changing state; TRUE alone does not mean fresh data.
AdsAddr is acyclic mailbox addressing information, not a measurement-validity indicator.
Select standard status-plus-value PDOs matching the declared Value type; compact value-only PDOs
are outside this model. Configure electrical range and scaling separately on the device.
</description>
*)
TYPE EL3051_EX EXTENDS EL3051 :
STRUCT
	WcState AT %I* : BOOL;
	InputToggle AT %I* : BOOL;
	State AT %I* : UINT;
	AdsAddr AT %I* : Global.AMSADDR;
END_STRUCT
END_TYPE

// ---- AnalogIO/Inputs/EL3052/EL3052.TcDUT
(*
SPDX-FileCopyrightText: © 2026 Oleksandr Tiutyk <trofimich@gmail.com>
SPDX-License-Identifier: MIT
License: https://opensource.org/license/mit
*)

(*!
<summary>
Beckhoff EL3052: 2-channel analog input terminal (4 .. 20 mA, 12-bit single-ended).
</summary>
<description>
Process image mapping structure for the EL3052 EtherCAT terminal with 2 analog input channel(s).
When used for I/O, link located fields or their containing buffers to the matching selected PDOs.
The record is not a packed wire buffer; compiler padding is not part of the device specification.
Unlinked/default values do not prove valid I/O. The caller evaluates bus/channel validity before use.
Use one owner task per instance and externally synchronize other access; multi-field snapshots are not atomic.
Copies store data without creating hardware links. Keep borrowed field references valid while consumers are bound.
This passive record performs no validation, synchronization, configuration or protocol advancement.
Select standard status-plus-value PDOs matching the declared Value type; compact value-only PDOs
are outside this model. Configure electrical range and scaling separately on the device.
</description>
*)
TYPE EL3052 :
STRUCT
	Ch1 : ANALOG_INPUT_INT_CHANNEL;
	Ch2 : ANALOG_INPUT_INT_CHANNEL;
END_STRUCT
END_TYPE

// ---- AnalogIO/Inputs/EL3052/EL3052_EX.TcDUT
(*
SPDX-FileCopyrightText: © 2026 Oleksandr Tiutyk <trofimich@gmail.com>
SPDX-License-Identifier: MIT
License: https://opensource.org/license/mit
*)

(*!
<summary>
Beckhoff EL3052_EX: Extended 2-channel analog input terminal (4 .. 20 mA, 12-bit single-ended) with
diagnostics.
</summary>
<description>
Extends EL3052 with EtherCAT Working Counter, slave state, and CoE mailbox ADS address diagnostics.
When used for I/O, link located fields or their containing buffers to the matching selected PDOs.
The record is not a packed wire buffer; compiler padding is not part of the device specification.
Unlinked/default values do not prove valid I/O. The caller evaluates bus/channel validity before use.
Use one owner task per instance and externally synchronize other access; multi-field snapshots are not atomic.
Copies store data without creating hardware links. Keep borrowed field references valid while consumers are bound.
This passive record performs no validation, synchronization, configuration or protocol advancement.
WcState=TRUE means process-data exchange is invalid. State is acyclic EtherCAT/link information,
not proof of current measurement validity. Link diagnostics to the matching slave InfoData entries.
The selected PDO representation is documented by the base terminal model.
InputToggle signals an input update by changing state; TRUE alone does not mean fresh data.
AdsAddr is acyclic mailbox addressing information, not a measurement-validity indicator.
Select standard status-plus-value PDOs matching the declared Value type; compact value-only PDOs
are outside this model. Configure electrical range and scaling separately on the device.
</description>
*)
TYPE EL3052_EX EXTENDS EL3052 :
STRUCT
	WcState AT %I* : BOOL;
	InputToggle AT %I* : BOOL;
	State AT %I* : UINT;
	AdsAddr AT %I* : Global.AMSADDR;
END_STRUCT
END_TYPE

// ---- AnalogIO/Inputs/EL3054/EL3054.TcDUT
(*
SPDX-FileCopyrightText: © 2026 Oleksandr Tiutyk <trofimich@gmail.com>
SPDX-License-Identifier: MIT
License: https://opensource.org/license/mit
*)

(*!
<summary>
Beckhoff EL3054: 4-channel analog input terminal (4 .. 20 mA, 12-bit single-ended).
</summary>
<description>
Process image mapping structure for the EL3054 EtherCAT terminal with 4 analog input channel(s).
When used for I/O, link located fields or their containing buffers to the matching selected PDOs.
The record is not a packed wire buffer; compiler padding is not part of the device specification.
Unlinked/default values do not prove valid I/O. The caller evaluates bus/channel validity before use.
Use one owner task per instance and externally synchronize other access; multi-field snapshots are not atomic.
Copies store data without creating hardware links. Keep borrowed field references valid while consumers are bound.
This passive record performs no validation, synchronization, configuration or protocol advancement.
Select standard status-plus-value PDOs matching the declared Value type; compact value-only PDOs
are outside this model. Configure electrical range and scaling separately on the device.
</description>
*)
TYPE EL3054 :
STRUCT
	Ch1 : ANALOG_INPUT_INT_CHANNEL;
	Ch2 : ANALOG_INPUT_INT_CHANNEL;
	Ch3 : ANALOG_INPUT_INT_CHANNEL;
	Ch4 : ANALOG_INPUT_INT_CHANNEL;
END_STRUCT
END_TYPE

// ---- AnalogIO/Inputs/EL3054/EL3054_EX.TcDUT
(*
SPDX-FileCopyrightText: © 2026 Oleksandr Tiutyk <trofimich@gmail.com>
SPDX-License-Identifier: MIT
License: https://opensource.org/license/mit
*)

(*!
<summary>
Beckhoff EL3054_EX: Extended 4-channel analog input terminal (4 .. 20 mA, 12-bit single-ended) with
diagnostics.
</summary>
<description>
Extends EL3054 with EtherCAT Working Counter, slave state, and CoE mailbox ADS address diagnostics.
When used for I/O, link located fields or their containing buffers to the matching selected PDOs.
The record is not a packed wire buffer; compiler padding is not part of the device specification.
Unlinked/default values do not prove valid I/O. The caller evaluates bus/channel validity before use.
Use one owner task per instance and externally synchronize other access; multi-field snapshots are not atomic.
Copies store data without creating hardware links. Keep borrowed field references valid while consumers are bound.
This passive record performs no validation, synchronization, configuration or protocol advancement.
WcState=TRUE means process-data exchange is invalid. State is acyclic EtherCAT/link information,
not proof of current measurement validity. Link diagnostics to the matching slave InfoData entries.
The selected PDO representation is documented by the base terminal model.
InputToggle signals an input update by changing state; TRUE alone does not mean fresh data.
AdsAddr is acyclic mailbox addressing information, not a measurement-validity indicator.
Select standard status-plus-value PDOs matching the declared Value type; compact value-only PDOs
are outside this model. Configure electrical range and scaling separately on the device.
</description>
*)
TYPE EL3054_EX EXTENDS EL3054 :
STRUCT
	WcState AT %I* : BOOL;
	InputToggle AT %I* : BOOL;
	State AT %I* : UINT;
	AdsAddr AT %I* : Global.AMSADDR;
END_STRUCT
END_TYPE

// ---- AnalogIO/Inputs/EL3058/EL3058.TcDUT
(*
SPDX-FileCopyrightText: © 2026 Oleksandr Tiutyk <trofimich@gmail.com>
SPDX-License-Identifier: MIT
License: https://opensource.org/license/mit
*)

(*!
<summary>
Beckhoff EL3058: 8-channel analog input terminal (4 .. 20 mA, 12-bit single-ended).
</summary>
<description>
Process image mapping structure for the EL3058 EtherCAT terminal with 8 analog input channel(s).
When used for I/O, link located fields or their containing buffers to the matching selected PDOs.
The record is not a packed wire buffer; compiler padding is not part of the device specification.
Unlinked/default values do not prove valid I/O. The caller evaluates bus/channel validity before use.
Use one owner task per instance and externally synchronize other access; multi-field snapshots are not atomic.
Copies store data without creating hardware links. Keep borrowed field references valid while consumers are bound.
This passive record performs no validation, synchronization, configuration or protocol advancement.
Select standard status-plus-value PDOs matching the declared Value type; compact value-only PDOs
are outside this model. Configure electrical range and scaling separately on the device.
</description>
*)
TYPE EL3058 :
STRUCT
	Ch1 : ANALOG_INPUT_INT_CHANNEL;
	Ch2 : ANALOG_INPUT_INT_CHANNEL;
	Ch3 : ANALOG_INPUT_INT_CHANNEL;
	Ch4 : ANALOG_INPUT_INT_CHANNEL;
	Ch5 : ANALOG_INPUT_INT_CHANNEL;
	Ch6 : ANALOG_INPUT_INT_CHANNEL;
	Ch7 : ANALOG_INPUT_INT_CHANNEL;
	Ch8 : ANALOG_INPUT_INT_CHANNEL;
END_STRUCT
END_TYPE

// ---- AnalogIO/Inputs/EL3058/EL3058_EX.TcDUT
(*
SPDX-FileCopyrightText: © 2026 Oleksandr Tiutyk <trofimich@gmail.com>
SPDX-License-Identifier: MIT
License: https://opensource.org/license/mit
*)

(*!
<summary>
Beckhoff EL3058_EX: Extended 8-channel analog input terminal (4 .. 20 mA, 12-bit single-ended) with
diagnostics.
</summary>
<description>
Extends EL3058 with EtherCAT Working Counter, slave state, and CoE mailbox ADS address diagnostics.
When used for I/O, link located fields or their containing buffers to the matching selected PDOs.
The record is not a packed wire buffer; compiler padding is not part of the device specification.
Unlinked/default values do not prove valid I/O. The caller evaluates bus/channel validity before use.
Use one owner task per instance and externally synchronize other access; multi-field snapshots are not atomic.
Copies store data without creating hardware links. Keep borrowed field references valid while consumers are bound.
This passive record performs no validation, synchronization, configuration or protocol advancement.
WcState=TRUE means process-data exchange is invalid. State is acyclic EtherCAT/link information,
not proof of current measurement validity. Link diagnostics to the matching slave InfoData entries.
The selected PDO representation is documented by the base terminal model.
InputToggle signals an input update by changing state; TRUE alone does not mean fresh data.
AdsAddr is acyclic mailbox addressing information, not a measurement-validity indicator.
Select standard status-plus-value PDOs matching the declared Value type; compact value-only PDOs
are outside this model. Configure electrical range and scaling separately on the device.
</description>
*)
TYPE EL3058_EX EXTENDS EL3058 :
STRUCT
	WcState AT %I* : BOOL;
	InputToggle AT %I* : BOOL;
	State AT %I* : UINT;
	AdsAddr AT %I* : Global.AMSADDR;
END_STRUCT
END_TYPE

// ---- AnalogIO/Inputs/EL3102/EL3102.TcDUT
(*
SPDX-FileCopyrightText: © 2026 Oleksandr Tiutyk <trofimich@gmail.com>
SPDX-License-Identifier: MIT
License: https://opensource.org/license/mit
*)

(*!
<summary>
Beckhoff EL3102: 2-channel analog input terminal (-10 V .. +10 V, 16-bit differential).
</summary>
<description>
Process image mapping structure for the EL3102 EtherCAT terminal with 2 analog input channel(s).
When used for I/O, link located fields or their containing buffers to the matching selected PDOs.
The record is not a packed wire buffer; compiler padding is not part of the device specification.
Unlinked/default values do not prove valid I/O. The caller evaluates bus/channel validity before use.
Use one owner task per instance and externally synchronize other access; multi-field snapshots are not atomic.
Copies store data without creating hardware links. Keep borrowed field references valid while consumers are bound.
This passive record performs no validation, synchronization, configuration or protocol advancement.
Select standard status-plus-value PDOs matching the declared Value type; compact value-only PDOs
are outside this model. Configure electrical range and scaling separately on the device.
</description>
*)
TYPE EL3102 :
STRUCT
	Ch1 : ANALOG_INPUT_INT_CHANNEL;
	Ch2 : ANALOG_INPUT_INT_CHANNEL;
END_STRUCT
END_TYPE

// ---- AnalogIO/Inputs/EL3102/EL3102_EX.TcDUT
(*
SPDX-FileCopyrightText: © 2026 Oleksandr Tiutyk <trofimich@gmail.com>
SPDX-License-Identifier: MIT
License: https://opensource.org/license/mit
*)

(*!
<summary>
Beckhoff EL3102_EX: Extended 2-channel analog input terminal (-10 V .. +10 V, 16-bit differential) with
diagnostics.
</summary>
<description>
Extends EL3102 with EtherCAT Working Counter, slave state, and CoE mailbox ADS address diagnostics.
When used for I/O, link located fields or their containing buffers to the matching selected PDOs.
The record is not a packed wire buffer; compiler padding is not part of the device specification.
Unlinked/default values do not prove valid I/O. The caller evaluates bus/channel validity before use.
Use one owner task per instance and externally synchronize other access; multi-field snapshots are not atomic.
Copies store data without creating hardware links. Keep borrowed field references valid while consumers are bound.
This passive record performs no validation, synchronization, configuration or protocol advancement.
WcState=TRUE means process-data exchange is invalid. State is acyclic EtherCAT/link information,
not proof of current measurement validity. Link diagnostics to the matching slave InfoData entries.
The selected PDO representation is documented by the base terminal model.
InputToggle signals an input update by changing state; TRUE alone does not mean fresh data.
AdsAddr is acyclic mailbox addressing information, not a measurement-validity indicator.
Select standard status-plus-value PDOs matching the declared Value type; compact value-only PDOs
are outside this model. Configure electrical range and scaling separately on the device.
</description>
*)
TYPE EL3102_EX EXTENDS EL3102 :
STRUCT
	WcState AT %I* : BOOL;
	InputToggle AT %I* : BOOL;
	State AT %I* : UINT;
	AdsAddr AT %I* : Global.AMSADDR;
END_STRUCT
END_TYPE

// ---- AnalogIO/Inputs/EL3104/EL3104.TcDUT
(*
SPDX-FileCopyrightText: © 2026 Oleksandr Tiutyk <trofimich@gmail.com>
SPDX-License-Identifier: MIT
License: https://opensource.org/license/mit
*)

(*!
<summary>
Beckhoff EL3104: 4-channel analog input terminal (-10 V .. +10 V, 16-bit differential).
</summary>
<description>
Process image mapping structure for the EL3104 EtherCAT terminal with 4 analog input channel(s).
When used for I/O, link located fields or their containing buffers to the matching selected PDOs.
The record is not a packed wire buffer; compiler padding is not part of the device specification.
Unlinked/default values do not prove valid I/O. The caller evaluates bus/channel validity before use.
Use one owner task per instance and externally synchronize other access; multi-field snapshots are not atomic.
Copies store data without creating hardware links. Keep borrowed field references valid while consumers are bound.
This passive record performs no validation, synchronization, configuration or protocol advancement.
Select standard status-plus-value PDOs matching the declared Value type; compact value-only PDOs
are outside this model. Configure electrical range and scaling separately on the device.
</description>
*)
TYPE EL3104 :
STRUCT
	Ch1 : ANALOG_INPUT_INT_CHANNEL;
	Ch2 : ANALOG_INPUT_INT_CHANNEL;
	Ch3 : ANALOG_INPUT_INT_CHANNEL;
	Ch4 : ANALOG_INPUT_INT_CHANNEL;
END_STRUCT
END_TYPE

// ---- AnalogIO/Inputs/EL3104/EL3104_EX.TcDUT
(*
SPDX-FileCopyrightText: © 2026 Oleksandr Tiutyk <trofimich@gmail.com>
SPDX-License-Identifier: MIT
License: https://opensource.org/license/mit
*)

(*!
<summary>
Beckhoff EL3104_EX: Extended 4-channel analog input terminal (-10 V .. +10 V, 16-bit differential) with
diagnostics.
</summary>
<description>
Extends EL3104 with EtherCAT Working Counter, slave state, and CoE mailbox ADS address diagnostics.
When used for I/O, link located fields or their containing buffers to the matching selected PDOs.
The record is not a packed wire buffer; compiler padding is not part of the device specification.
Unlinked/default values do not prove valid I/O. The caller evaluates bus/channel validity before use.
Use one owner task per instance and externally synchronize other access; multi-field snapshots are not atomic.
Copies store data without creating hardware links. Keep borrowed field references valid while consumers are bound.
This passive record performs no validation, synchronization, configuration or protocol advancement.
WcState=TRUE means process-data exchange is invalid. State is acyclic EtherCAT/link information,
not proof of current measurement validity. Link diagnostics to the matching slave InfoData entries.
The selected PDO representation is documented by the base terminal model.
InputToggle signals an input update by changing state; TRUE alone does not mean fresh data.
AdsAddr is acyclic mailbox addressing information, not a measurement-validity indicator.
Select standard status-plus-value PDOs matching the declared Value type; compact value-only PDOs
are outside this model. Configure electrical range and scaling separately on the device.
</description>
*)
TYPE EL3104_EX EXTENDS EL3104 :
STRUCT
	WcState AT %I* : BOOL;
	InputToggle AT %I* : BOOL;
	State AT %I* : UINT;
	AdsAddr AT %I* : Global.AMSADDR;
END_STRUCT
END_TYPE

// ---- AnalogIO/Inputs/EL3122/EL3122.TcDUT
(*
SPDX-FileCopyrightText: © 2026 Oleksandr Tiutyk <trofimich@gmail.com>
SPDX-License-Identifier: MIT
License: https://opensource.org/license/mit
*)

(*!
<summary>
Beckhoff EL3122: 2-channel analog input terminal (4 .. 20 mA, 16-bit differential).
</summary>
<description>
Process image mapping structure for the EL3122 EtherCAT terminal with 2 analog input channel(s).
When used for I/O, link located fields or their containing buffers to the matching selected PDOs.
The record is not a packed wire buffer; compiler padding is not part of the device specification.
Unlinked/default values do not prove valid I/O. The caller evaluates bus/channel validity before use.
Use one owner task per instance and externally synchronize other access; multi-field snapshots are not atomic.
Copies store data without creating hardware links. Keep borrowed field references valid while consumers are bound.
This passive record performs no validation, synchronization, configuration or protocol advancement.
Select standard status-plus-value PDOs matching the declared Value type; compact value-only PDOs
are outside this model. Configure electrical range and scaling separately on the device.
</description>
*)
TYPE EL3122 :
STRUCT
	Ch1 : ANALOG_INPUT_INT_CHANNEL;
	Ch2 : ANALOG_INPUT_INT_CHANNEL;
END_STRUCT
END_TYPE

// ---- AnalogIO/Inputs/EL3122/EL3122_EX.TcDUT
(*
SPDX-FileCopyrightText: © 2026 Oleksandr Tiutyk <trofimich@gmail.com>
SPDX-License-Identifier: MIT
License: https://opensource.org/license/mit
*)

(*!
<summary>
Beckhoff EL3122_EX: Extended 2-channel analog input terminal (4 .. 20 mA, 16-bit differential) with
diagnostics.
</summary>
<description>
Extends EL3122 with EtherCAT Working Counter, slave state, and CoE mailbox ADS address diagnostics.
When used for I/O, link located fields or their containing buffers to the matching selected PDOs.
The record is not a packed wire buffer; compiler padding is not part of the device specification.
Unlinked/default values do not prove valid I/O. The caller evaluates bus/channel validity before use.
Use one owner task per instance and externally synchronize other access; multi-field snapshots are not atomic.
Copies store data without creating hardware links. Keep borrowed field references valid while consumers are bound.
This passive record performs no validation, synchronization, configuration or protocol advancement.
WcState=TRUE means process-data exchange is invalid. State is acyclic EtherCAT/link information,
not proof of current measurement validity. Link diagnostics to the matching slave InfoData entries.
The selected PDO representation is documented by the base terminal model.
InputToggle signals an input update by changing state; TRUE alone does not mean fresh data.
AdsAddr is acyclic mailbox addressing information, not a measurement-validity indicator.
Select standard status-plus-value PDOs matching the declared Value type; compact value-only PDOs
are outside this model. Configure electrical range and scaling separately on the device.
</description>
*)
TYPE EL3122_EX EXTENDS EL3122 :
STRUCT
	WcState AT %I* : BOOL;
	InputToggle AT %I* : BOOL;
	State AT %I* : UINT;
	AdsAddr AT %I* : Global.AMSADDR;
END_STRUCT
END_TYPE

// ---- AnalogIO/Inputs/EL3124/EL3124.TcDUT
(*
SPDX-FileCopyrightText: © 2026 Oleksandr Tiutyk <trofimich@gmail.com>
SPDX-License-Identifier: MIT
License: https://opensource.org/license/mit
*)

(*!
<summary>
Beckhoff EL3124: 4-channel analog input terminal (4 .. 20 mA, 16-bit differential).
</summary>
<description>
Process image mapping structure for the EL3124 EtherCAT terminal with 4 analog input channel(s).
When used for I/O, link located fields or their containing buffers to the matching selected PDOs.
The record is not a packed wire buffer; compiler padding is not part of the device specification.
Unlinked/default values do not prove valid I/O. The caller evaluates bus/channel validity before use.
Use one owner task per instance and externally synchronize other access; multi-field snapshots are not atomic.
Copies store data without creating hardware links. Keep borrowed field references valid while consumers are bound.
This passive record performs no validation, synchronization, configuration or protocol advancement.
Select standard status-plus-value PDOs matching the declared Value type; compact value-only PDOs
are outside this model. Configure electrical range and scaling separately on the device.
</description>
*)
TYPE EL3124 :
STRUCT
	Ch1 : ANALOG_INPUT_INT_CHANNEL;
	Ch2 : ANALOG_INPUT_INT_CHANNEL;
	Ch3 : ANALOG_INPUT_INT_CHANNEL;
	Ch4 : ANALOG_INPUT_INT_CHANNEL;
END_STRUCT
END_TYPE

// ---- AnalogIO/Inputs/EL3124/EL3124_EX.TcDUT
(*
SPDX-FileCopyrightText: © 2026 Oleksandr Tiutyk <trofimich@gmail.com>
SPDX-License-Identifier: MIT
License: https://opensource.org/license/mit
*)

(*!
<summary>
Beckhoff EL3124_EX: Extended 4-channel analog input terminal (4 .. 20 mA, 16-bit differential) with
diagnostics.
</summary>
<description>
Extends EL3124 with EtherCAT Working Counter, slave state, and CoE mailbox ADS address diagnostics.
When used for I/O, link located fields or their containing buffers to the matching selected PDOs.
The record is not a packed wire buffer; compiler padding is not part of the device specification.
Unlinked/default values do not prove valid I/O. The caller evaluates bus/channel validity before use.
Use one owner task per instance and externally synchronize other access; multi-field snapshots are not atomic.
Copies store data without creating hardware links. Keep borrowed field references valid while consumers are bound.
This passive record performs no validation, synchronization, configuration or protocol advancement.
WcState=TRUE means process-data exchange is invalid. State is acyclic EtherCAT/link information,
not proof of current measurement validity. Link diagnostics to the matching slave InfoData entries.
The selected PDO representation is documented by the base terminal model.
InputToggle signals an input update by changing state; TRUE alone does not mean fresh data.
AdsAddr is acyclic mailbox addressing information, not a measurement-validity indicator.
Select standard status-plus-value PDOs matching the declared Value type; compact value-only PDOs
are outside this model. Configure electrical range and scaling separately on the device.
</description>
*)
TYPE EL3124_EX EXTENDS EL3124 :
STRUCT
	WcState AT %I* : BOOL;
	InputToggle AT %I* : BOOL;
	State AT %I* : UINT;
	AdsAddr AT %I* : Global.AMSADDR;
END_STRUCT
END_TYPE

// ---- AnalogIO/Outputs/EL4021/EL4021.TcDUT
(*
SPDX-FileCopyrightText: © 2026 Oleksandr Tiutyk <trofimich@gmail.com>
SPDX-License-Identifier: MIT
License: https://opensource.org/license/mit
*)

(*!
<summary>
Beckhoff EL4021: 1-channel analog output terminal (4 .. 20 mA, 12-bit).
</summary>
<description>
Process image mapping structure for the EL4021 EtherCAT terminal with 1 analog output channel(s).
When used for I/O, link located fields or their containing buffers to the matching selected PDOs.
The record is not a packed wire buffer; compiler padding is not part of the device specification.
Unlinked/default values do not prove valid I/O. The caller evaluates bus/channel validity before use.
Use one owner task per instance and externally synchronize other access; multi-field snapshots are not atomic.
Copies store data without creating hardware links. Keep borrowed field references valid while consumers are bound.
This passive record performs no validation, synchronization, configuration or protocol advancement.
Channels hold raw INT16 output commands; configure electrical range and presentation before use.
</description>
*)
TYPE EL4021 :
STRUCT
	Ch1 AT %Q* : INT;
END_STRUCT
END_TYPE

// ---- AnalogIO/Outputs/EL4021/EL4021_EX.TcDUT
(*
SPDX-FileCopyrightText: © 2026 Oleksandr Tiutyk <trofimich@gmail.com>
SPDX-License-Identifier: MIT
License: https://opensource.org/license/mit
*)

(*!
<summary>
Beckhoff EL4021_EX: Extended 1-channel analog output terminal (4 .. 20 mA, 12-bit) with diagnostics.
</summary>
<description>
Extends EL4021 with EtherCAT Working Counter, slave state, and CoE mailbox ADS address diagnostics.
When used for I/O, link located fields or their containing buffers to the matching selected PDOs.
The record is not a packed wire buffer; compiler padding is not part of the device specification.
Unlinked/default values do not prove valid I/O. The caller evaluates bus/channel validity before use.
Use one owner task per instance and externally synchronize other access; multi-field snapshots are not atomic.
Copies store data without creating hardware links. Keep borrowed field references valid while consumers are bound.
This passive record performs no validation, synchronization, configuration or protocol advancement.
WcState=TRUE means process-data exchange is invalid. State is acyclic EtherCAT/link information,
not proof of current measurement validity. Link diagnostics to the matching slave InfoData entries.
The selected PDO representation is documented by the base terminal model.
AdsAddr is acyclic mailbox addressing information, not a measurement-validity indicator.
Channels hold raw INT16 output commands; configure electrical range and presentation before use.
</description>
*)
TYPE EL4021_EX EXTENDS EL4021 :
STRUCT
	WcState AT %I* : BOOL;
	State AT %I* : UINT;
	AdsAddr AT %I* : Global.AMSADDR;
END_STRUCT
END_TYPE

// ---- AnalogIO/Outputs/EL4022/EL4022.TcDUT
(*
SPDX-FileCopyrightText: © 2026 Oleksandr Tiutyk <trofimich@gmail.com>
SPDX-License-Identifier: MIT
License: https://opensource.org/license/mit
*)

(*!
<summary>
Beckhoff EL4022: 2-channel analog output terminal (4 .. 20 mA, 12-bit).
</summary>
<description>
Process image mapping structure for the EL4022 EtherCAT terminal with 2 analog output channel(s).
When used for I/O, link located fields or their containing buffers to the matching selected PDOs.
The record is not a packed wire buffer; compiler padding is not part of the device specification.
Unlinked/default values do not prove valid I/O. The caller evaluates bus/channel validity before use.
Use one owner task per instance and externally synchronize other access; multi-field snapshots are not atomic.
Copies store data without creating hardware links. Keep borrowed field references valid while consumers are bound.
This passive record performs no validation, synchronization, configuration or protocol advancement.
Channels hold raw INT16 output commands; configure electrical range and presentation before use.
</description>
*)
TYPE EL4022 :
STRUCT
	Ch1 AT %Q* : INT;
	Ch2 AT %Q* : INT;
END_STRUCT
END_TYPE

